FUNCTION_BLOCK BLOW_DOW_SEQ
VAR_IN_OUT
	xExecute:		BOOL;
	xDone:			BOOL;
END_VAR
VAR_OUTPUT
	
END_VAR
VAR
	tpReset:			TP;
	rtDone:				R_TRIG;
	rtExecute:			R_TRIG;
	ftTimePulse:		F_TRIG;
	tpTimePulse:		TP;
	lrTargetPos:		LREAL;
	xTransCondition:	BOOL;	
	xTransRelease:		BOOL;
	SFCInit:			BOOL;
	SFCReset:			BOOL;	
	SFCError:			BOOL;
END_VAR

rtDone(CLK:=xDone);
IF rtDone.Q THEN
	xTransRelease:=FALSE;	
	SFCReset:=TRUE;
	xExecute:=FALSE;
END_IF

rtExecute(CLK:=xExecute);
IF rtExecute.Q THEN
	xTransRelease:=TRUE;
END_IF

aSEQ_ACT();

tpReset(IN:=SFCError, PT:=T#250MS);
SFCReset:= tpReset.Q;

ACTION ACK_DONE_AXIS_active:
IF G_sAxisDone.X OR G_sAxisDone.Y OR G_sAxisDone.Z OR G_sAxisDone.c THEN
	G_sAckAxisDone.X:=TRUE;
	G_sAckAxisDone.Y:=TRUE;
	G_sAckAxisDone.Z:=TRUE;
	G_sAckAxisDone.C:=TRUE;
ELSE
	G_sAckAxisDone.X:=FALSE;
	G_sAckAxisDone.Y:=FALSE;
	G_sAckAxisDone.Z:=FALSE;
	G_sAckAxisDone.C:=FALSE;
END_IF

xTransCondition:= NOT G_sAckAxisDone.X AND NOT G_sAckAxisDone.Y AND NOT G_sAckAxisDone.Z AND NOT G_sAckAxisDone.C;
END_ACTION

ACTION aSEQ_ACT:
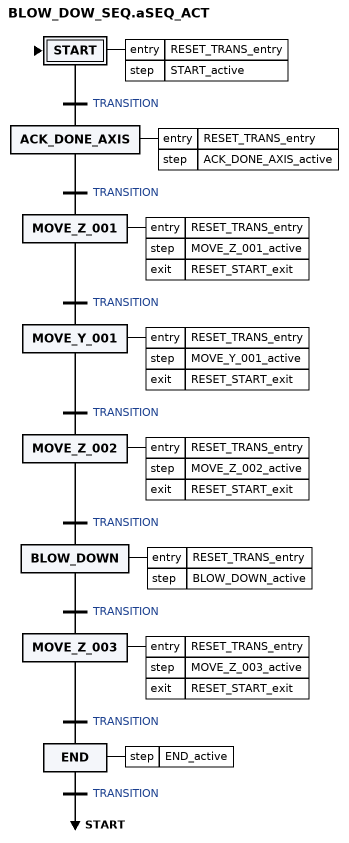
INITIAL_STEP START:
    RESET_TRANS_entry(P1);  // entry action
    START_active(N);  // step action
END_STEP
TRANSITION FROM START TO ACK_DONE_AXIS
    := TRANSITION;
END_TRANSITION
STEP ACK_DONE_AXIS:
    RESET_TRANS_entry(P1);  // entry action
    ACK_DONE_AXIS_active(N);  // step action
END_STEP
TRANSITION FROM ACK_DONE_AXIS TO MOVE_Z_001
    := TRANSITION;
END_TRANSITION
STEP MOVE_Z_001:
    RESET_TRANS_entry(P1);  // entry action
    MOVE_Z_001_active(N);  // step action
    RESET_START_exit(P0);  // exit action
END_STEP
TRANSITION FROM MOVE_Z_001 TO MOVE_Y_001
    := TRANSITION;
END_TRANSITION
STEP MOVE_Y_001:
    RESET_TRANS_entry(P1);  // entry action
    MOVE_Y_001_active(N);  // step action
    RESET_START_exit(P0);  // exit action
END_STEP
TRANSITION FROM MOVE_Y_001 TO MOVE_Z_002
    := TRANSITION;
END_TRANSITION
STEP MOVE_Z_002:
    RESET_TRANS_entry(P1);  // entry action
    MOVE_Z_002_active(N);  // step action
    RESET_START_exit(P0);  // exit action
END_STEP
TRANSITION FROM MOVE_Z_002 TO BLOW_DOWN
    := TRANSITION;
END_TRANSITION
STEP BLOW_DOWN:
    RESET_TRANS_entry(P1);  // entry action
    BLOW_DOWN_active(N);  // step action
END_STEP
TRANSITION FROM BLOW_DOWN TO MOVE_Z_003
    := TRANSITION;
END_TRANSITION
STEP MOVE_Z_003:
    RESET_TRANS_entry(P1);  // entry action
    MOVE_Z_003_active(N);  // step action
    RESET_START_exit(P0);  // exit action
END_STEP
TRANSITION FROM MOVE_Z_003 TO END
    := TRANSITION;
END_TRANSITION
STEP END:
    END_active(N);  // step action
END_STEP
TRANSITION FROM END TO START
    := TRANSITION;
END_TRANSITION
END_ACTION

ACTION BLOW_DOWN_active:
tpTimePulse(IN:=NOT tpTimePulse.Q, PT:=T#3000MS);
ftTimePulse(CLK:=tpTimePulse.Q);
xTransCondition:= ftTimePulse.Q;
END_ACTION

ACTION END_active:
xDone:=TRUE;
xTransCondition:=xDone;
END_ACTION

ACTION MOVE_Y_001_active:
G_sTargetPosition.Y:= G_asIndividualAxisPositions[CE_AXIS_Y].Positions[1].Target;
G_sStartToPos.Y:= TRUE;

xTransCondition:= G_sAxisDone.Y;
END_ACTION

ACTION MOVE_Z_001_active:
G_sTargetPosition.Z:= G_asIndividualAxisPositions[CE_AXIS_Z].Positions[1].Target;
G_sStartToPos.Z:= TRUE;

xTransCondition:= G_sAxisDone.Z;
END_ACTION

ACTION MOVE_Z_002_active:
G_sTargetPosition.Z:= G_asIndividualAxisPositions[CE_AXIS_Z].Positions[2].Target;
G_sStartToPos.Z:= TRUE;

xTransCondition:= G_sAxisDone.Z;
END_ACTION

ACTION MOVE_Z_003_active:
G_sTargetPosition.Z:= G_asIndividualAxisPositions[CE_AXIS_Z].Positions[1].Target;
G_sStartToPos.Z:= TRUE;

xTransCondition:= G_sAxisDone.Z;
END_ACTION

ACTION RESET_START_exit:
IF G_sAxisDone.X OR G_sAxisDone.Y OR G_sAxisDone.Z OR G_sAxisDone.c THEN
	G_sAckAxisDone.X:=TRUE;
	G_sAckAxisDone.Y:=TRUE;
	G_sAckAxisDone.Z:=TRUE;
	G_sAckAxisDone.C:=TRUE;
ELSE
	G_sAckAxisDone.X:=FALSE;
	G_sAckAxisDone.Y:=FALSE;
	G_sAckAxisDone.Z:=FALSE;
	G_sAckAxisDone.C:=FALSE;
	
	G_sStartToPos.X:=FALSE;
	G_sStartToPos.Y:=FALSE;
	G_sStartToPos.Z:=FALSE;
	G_sStartToPos.C:=FALSE;
END_IF
END_ACTION

ACTION RESET_TRANS_entry:
xTransCondition:= false;
END_ACTION

ACTION START_active:
xDone:=FALSE;
xTransCondition:= NOT xDone;
END_ACTION

TRANSITION TRANSITION:
xTransRelease AND xTransCondition
END_TRANSITION

END_FUNCTION_BLOCK

(* stored: Version 1.1.0.1, ProductVersion 3.1.4022.18
   POU BLOW_DOW_SEQ: Id {cf72467f-b60c-43e5-909f-e1d6bfbab1c5}, SpecialFunc None
   Folder xActive: Id {94637cd7-7d63-4c1f-af4b-ab4b9dbff51c}
   Folder xEntry: Id {c57fb69f-dfbe-4344-b0fa-99be7f007b87}
   Folder xExit: Id {c667e7ae-4ce1-40fe-acc9-2ca912cf4588}
   Folder xTrans: Id {519adcc3-a82c-48fe-ae37-052122a02f8d}
   Action ACK_DONE_AXIS_active: Id {9fc1dd64-3186-4599-84f6-d0ff90917ad0}
   Action aSEQ_ACT: Id {a78325bd-2dbb-432d-a1ad-92d0e473dbbf}
   Action BLOW_DOWN_active: Id {54c4b2b1-1a1f-48ef-ad85-4730ca13d443}
   Action END_active: Id {43cdd48b-c7d6-43c4-96c3-5db2a321ac7a}
   Action MOVE_Y_001_active: Id {24cb28b6-d1a1-4ed1-8316-eea14b0be8e3}
   Action MOVE_Z_001_active: Id {9744347d-9b2b-445a-9369-5c38b13c2f56}
   Action MOVE_Z_002_active: Id {cc97c7bc-2bb3-495d-8a11-4743d6ee7c59}
   Action MOVE_Z_003_active: Id {99f11d0d-a2bc-4119-909b-061f1fe4583a}
   Action RESET_START_exit: Id {23faa2d5-a3d8-4b9d-9ca5-8fe226ddf9f4}
   Action RESET_TRANS_entry: Id {47b00800-ab98-4932-ad3f-cb8a7cd213ce}
   Action START_active: Id {638bbd12-e889-4e3e-8e45-f0e4a52a0bff}
   Transition TRANSITION: Id {7541fc43-f12d-4744-b161-15076261fd7e} *)
